PROGRAM MAIN
VAR
	fb_Measurement1: FB_Measurement;
	fb_Measurement2: FB_Measurement;
	fb_Measurement3: FB_Measurement;
	fb_Measurement4: FB_Measurement;
	fb_Measurement5: FB_Measurement;
	fb_Measurement6: FB_Measurement;
	fb_Measurement7: FB_Measurement;
	fb_Measurement8: FB_Measurement;
	fb_Measurement9: FB_Measurement;
	fb_Measurement10: FB_Measurement;
END_VAR

fb_Measurement1(
	// Measurement settings
	nHighLevel:=20, 
	nLowLevel:=5 ,
	nHighDuration:=T#5S, 
	nLowDuration:=T#5S,
	nRandomizerSeedValue := 10, 
	delayTimeAfterAddOrSub :=T#1000MS,
	nStepValueMult :=1,
	// Measurement value
	nMeasValue=>GVL.nMeasurement1);
	
fb_Measurement2(
	nHighLevel:=30, 
	nLowLevel:=-30, 
	nHighDuration:=T#5S, 
	nLowDuration:=T#5S,
	nRandomizerSeedValue := 7, 
	delayTimeAfterAddOrSub :=T#1000MS,
	nStepValueMult :=0.1,
	nMeasValue=>GVL.nMeasurement2);
	
fb_Measurement3(
	nHighLevel:=-1, 
	nLowLevel:=-7, 
	nHighDuration:=T#5S, 
	nLowDuration:=T#5S,
	nRandomizerSeedValue := 42, 
	delayTimeAfterAddOrSub :=T#1000MS,
	nStepValueMult :=0.01,
	nMeasValue=>GVL.nMeasurement3);

fb_Measurement4(
    nHighLevel:=10, 
    nLowLevel:=-10, 
    nHighDuration:=T#5S, 
    nLowDuration:=T#5S, 
    nRandomizerSeedValue:=5, 
    delayTimeAfterAddOrSub:=T#1000MS, 
    nStepValueMult:=0.2, 
    nMeasValue=>GVL.nMeasurement4);

fb_Measurement5(
    nHighLevel:=15, 
    nLowLevel:=-5, 
    nHighDuration:=T#5S, 
    nLowDuration:=T#5S, 
    nRandomizerSeedValue:=25, 
    delayTimeAfterAddOrSub:=T#1000MS, 
    nStepValueMult:=0.15, 
    nMeasValue=>GVL.nMeasurement5);

fb_Measurement6(
    nHighLevel:=5, 
    nLowLevel:=-10, 
    nHighDuration:=T#5S, 
    nLowDuration:=T#5S, 
    nRandomizerSeedValue:=30, 
    delayTimeAfterAddOrSub:=T#1000MS, 
    nStepValueMult:=0.05, 
    nMeasValue=>GVL.nMeasurement6);

fb_Measurement7(
    nHighLevel:=20, 
    nLowLevel:=10, 
    nHighDuration:=T#5S, 
    nLowDuration:=T#5S, 
    nRandomizerSeedValue:=35, 
    delayTimeAfterAddOrSub:=T#1000MS, 
    nStepValueMult:=0.25, 
    nMeasValue=>GVL.nMeasurement7);

fb_Measurement8(
    nHighLevel:=25, 
    nLowLevel:=-15, 
    nHighDuration:=T#5S, 
    nLowDuration:=T#5S, 
    nRandomizerSeedValue:=45, 
    delayTimeAfterAddOrSub:=T#1000MS, 
    nStepValueMult:=0.1, 
    nMeasValue=>GVL.nMeasurement8);

fb_Measurement9(
    nHighLevel:=-5, 
    nLowLevel:=-20, 
    nHighDuration:=T#5S, 
    nLowDuration:=T#5S, 
    nRandomizerSeedValue:=50, 
    delayTimeAfterAddOrSub:=T#1000MS, 
    nStepValueMult:=0.02, 
    nMeasValue=>GVL.nMeasurement9);

fb_Measurement10(
    nHighLevel:=12, 
    nLowLevel:=-8, 
    nHighDuration:=T#5S, 
    nLowDuration:=T#5S, 
    nRandomizerSeedValue:=60, 
    delayTimeAfterAddOrSub:=T#1000MS, 
    nStepValueMult:=0.12, 
    nMeasValue=>GVL.nMeasurement10);

END_PROGRAM

(* stored: Version 1.1.0.1, ProductVersion 3.1.4026.8
   POU MAIN: Id {2af31032-8259-45cf-8681-dab57608e6fa}, SpecialFunc None *)
